PROGRAM STN_TopUpCtrl
VAR

END_VAR

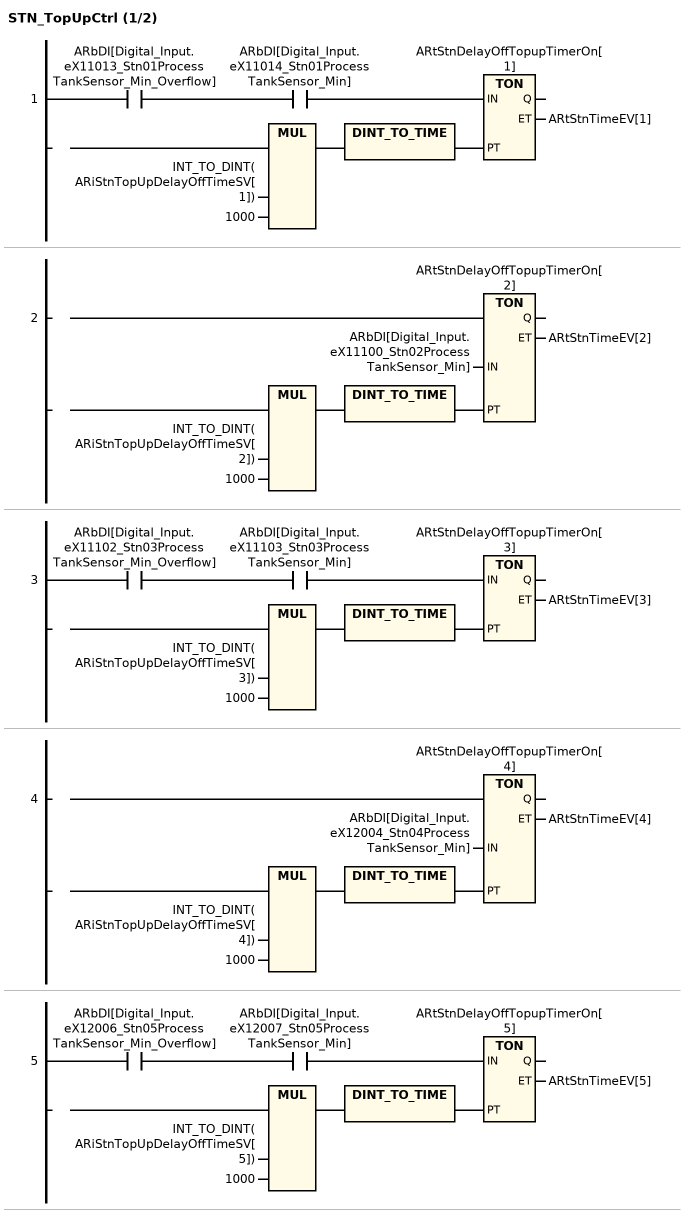
// NETWORK 1
ARtStnDelayOffTopupTimerOn[1](
    IN := ARbDI[Digital_Input.eX11013_Stn01ProcessTankSensor_Min_Overflow] AND ARbDI[Digital_Input.eX11014_Stn01ProcessTankSensor_Min],
    PT := DINT_TO_TIME((INT_TO_DINT(ARiStnTopUpDelayOffTimeSV[1])) * 1000),
    ET => ARtStnTimeEV[1]); // TON

// NETWORK 2
ARtStnDelayOffTopupTimerOn[2](
    IN := ARbDI[Digital_Input.eX11100_Stn02ProcessTankSensor_Min],
    PT := DINT_TO_TIME((INT_TO_DINT(ARiStnTopUpDelayOffTimeSV[2])) * 1000),
    ET => ARtStnTimeEV[2]); // TON

// NETWORK 3
ARtStnDelayOffTopupTimerOn[3](
    IN := ARbDI[Digital_Input.eX11102_Stn03ProcessTankSensor_Min_Overflow] AND ARbDI[Digital_Input.eX11103_Stn03ProcessTankSensor_Min],
    PT := DINT_TO_TIME((INT_TO_DINT(ARiStnTopUpDelayOffTimeSV[3])) * 1000),
    ET => ARtStnTimeEV[3]); // TON

// NETWORK 4
ARtStnDelayOffTopupTimerOn[4](
    IN := ARbDI[Digital_Input.eX12004_Stn04ProcessTankSensor_Min],
    PT := DINT_TO_TIME((INT_TO_DINT(ARiStnTopUpDelayOffTimeSV[4])) * 1000),
    ET => ARtStnTimeEV[4]); // TON

// NETWORK 5
ARtStnDelayOffTopupTimerOn[5](
    IN := ARbDI[Digital_Input.eX12006_Stn05ProcessTankSensor_Min_Overflow] AND ARbDI[Digital_Input.eX12007_Stn05ProcessTankSensor_Min],
    PT := DINT_TO_TIME((INT_TO_DINT(ARiStnTopUpDelayOffTimeSV[5])) * 1000),
    ET => ARtStnTimeEV[5]); // TON

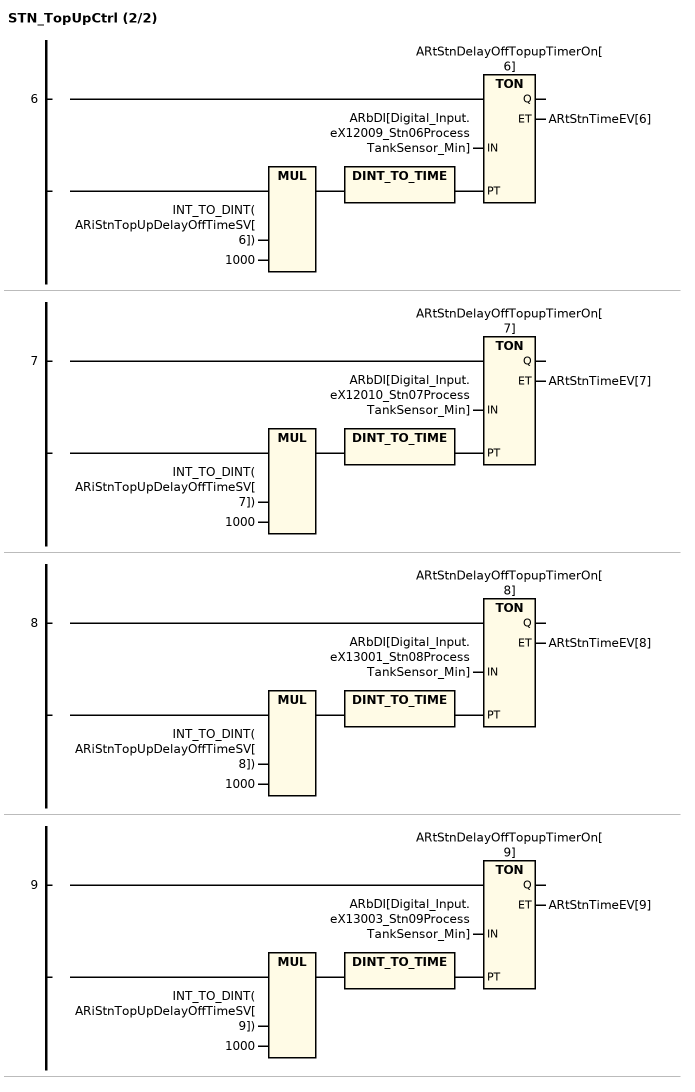
// NETWORK 6
ARtStnDelayOffTopupTimerOn[6](
    IN := ARbDI[Digital_Input.eX12009_Stn06ProcessTankSensor_Min],
    PT := DINT_TO_TIME((INT_TO_DINT(ARiStnTopUpDelayOffTimeSV[6])) * 1000),
    ET => ARtStnTimeEV[6]); // TON

// NETWORK 7
ARtStnDelayOffTopupTimerOn[7](
    IN := ARbDI[Digital_Input.eX12010_Stn07ProcessTankSensor_Min],
    PT := DINT_TO_TIME((INT_TO_DINT(ARiStnTopUpDelayOffTimeSV[7])) * 1000),
    ET => ARtStnTimeEV[7]); // TON

// NETWORK 8
ARtStnDelayOffTopupTimerOn[8](
    IN := ARbDI[Digital_Input.eX13001_Stn08ProcessTankSensor_Min],
    PT := DINT_TO_TIME((INT_TO_DINT(ARiStnTopUpDelayOffTimeSV[8])) * 1000),
    ET => ARtStnTimeEV[8]); // TON

// NETWORK 9
ARtStnDelayOffTopupTimerOn[9](
    IN := ARbDI[Digital_Input.eX13003_Stn09ProcessTankSensor_Min],
    PT := DINT_TO_TIME((INT_TO_DINT(ARiStnTopUpDelayOffTimeSV[9])) * 1000),
    ET => ARtStnTimeEV[9]); // TON

END_PROGRAM

(* stored: Version 1.1.0.1, ProductVersion 3.1.4024.12
   POU STN_TopUpCtrl: Id {2796cbd1-2e75-492e-a20f-393c17b7d8b3}, SpecialFunc None *)
